{attribute 'qualified_only'}
VAR_GLOBAL
	iTaskIdx 	: DINT;
	bFirstCycle : BOOL;
END_VAR

(* stored: Version 1.1.0.1, ProductVersion 3.1.4024.12
   GVL PLCSystem: Id {4f95d190-3ef4-4290-bb7f-6ba46402401b} *)
